(* Schneider Machine Expert - Basic project Timer New, file version 1.7.0.0 *)
(* ProjectInformations: Name=New project *)

HARDWARE
  Cpu 0: TM221M16R/G
  EthernetConfiguration: NetworkName=M221, IpAllocationMode=FixedAddress, IpAddress=0.0.0.0, SubnetMask=0.0.0.0
  SerialLineConfiguration: Baud=Baud19200, Parity=ParityEven, DataBits=DataBits8, StopBits=StopBits1, PhysicalMedium=PhysicalMediumRs485, TransmissionMode=TransmissionModeModbusRtu, SlaveId=1, Addressing=SlaveAddressing
  MastTask: UsePeriodScanMode=false, PeriodScan=100
  FastTask: Period=255
  CpuBehavior: StartingMode=StartAsPreviousState, AutoSaveRamOnEeprom=true, WatchdogPeriod=250

SYMBOLS  (address, symbol, comment, settings)
  %TM0        "T1"  [Preset=1, Base=OneSecond]
  %TM1        "T2"  [Preset=1, Base=OneSecond]
  %TM2        "T3"  [Preset=1, Base=OneSecond]
  %TM3        "T4"  [Preset=1, Base=OneSecond]
  %TM4        "TM5"  [Preset=1, Base=OneSecond]
  %TM5        "TM6"  [Preset=1, Base=OneSecond]
  %TM6        "TM7"  [Preset=1, Base=OneSecond]
  %TM7        "T8"  [Preset=1, Base=OneSecond]
  %I0.0       "Auto"
  %Q0.0       "L1"
  %Q0.1       "L2"
  %Q0.2       "L3"
  %Q0.3       "L4"

POU New POU
  (* SectionNumber=1 *)

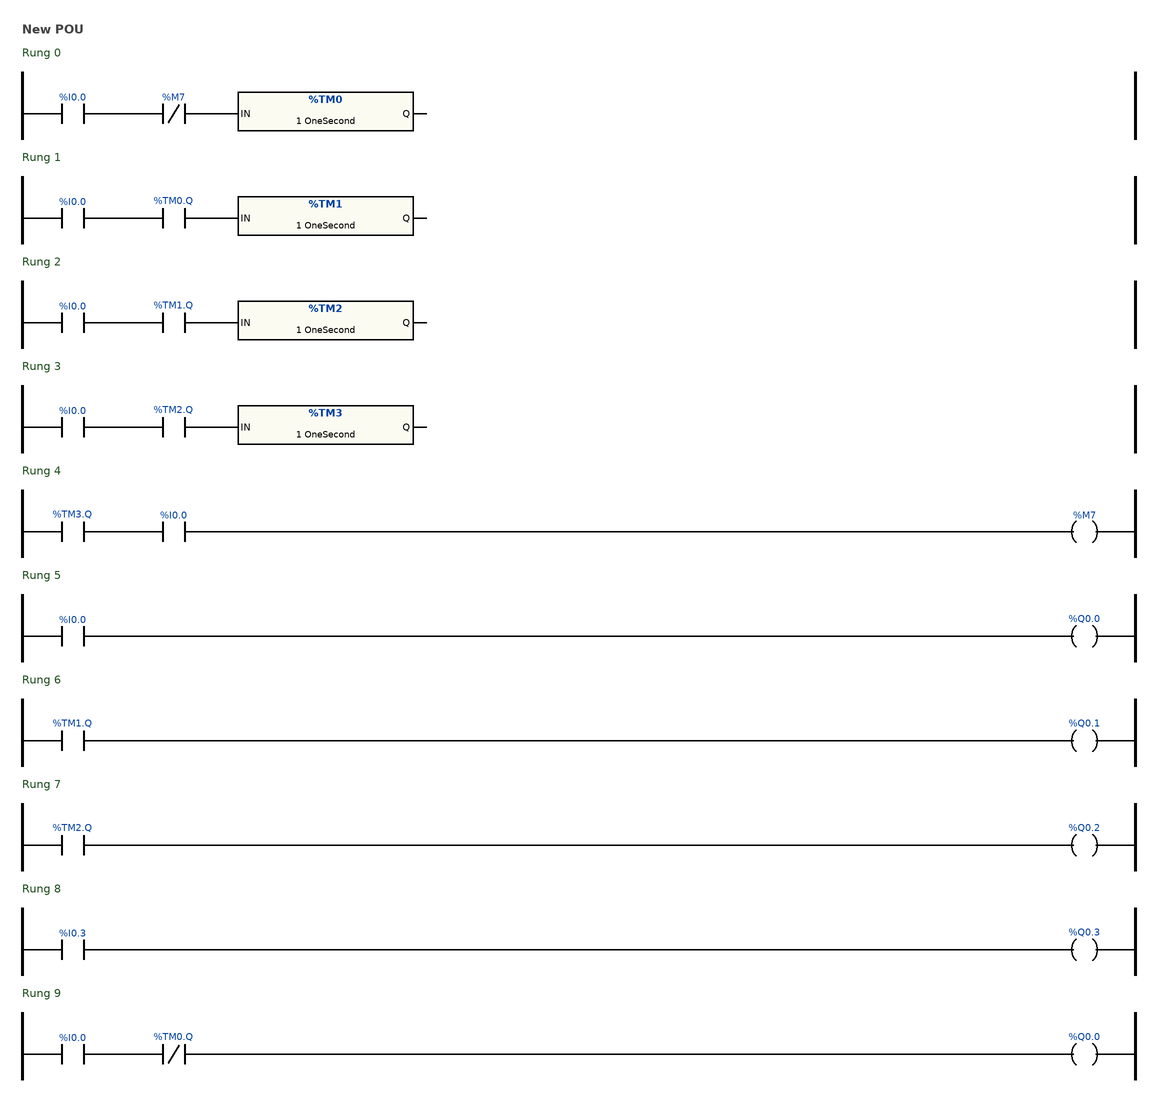

// Rung 0
  BLK %TM0
  LD %I0.0
  ANDN %M7
  IN
  END_BLK
  // as ST:
  //   %TM0(IN := %I0.0 AND NOT %M7);

// Rung 1
  BLK %TM1
  LD %I0.0
  AND %TM0.Q
  IN
  END_BLK
  // as ST:
  //   %TM1(IN := %I0.0 AND %TM0.Q);

// Rung 2
  BLK %TM2
  LD %I0.0
  AND %TM1.Q
  IN
  END_BLK
  // as ST:
  //   %TM2(IN := %I0.0 AND %TM1.Q);

// Rung 3
  BLK %TM3
  LD %I0.0
  AND %TM2.Q
  IN
  END_BLK
  // as ST:
  //   %TM3(IN := %I0.0 AND %TM2.Q);

// Rung 4
  LD %TM3.Q
  AND %I0.0
  ST %M7
  // as ST:
  //   %M7 := %TM3.Q AND %I0.0;

// Rung 5
  LD %I0.0
  ST %Q0.0
  // as ST:
  //   %Q0.0 := %I0.0;

// Rung 6
  LD %TM1.Q
  ST %Q0.1
  // as ST:
  //   %Q0.1 := %TM1.Q;

// Rung 7
  LD %TM2.Q
  ST %Q0.2
  // as ST:
  //   %Q0.2 := %TM2.Q;

// Rung 8
  LD %I0.3
  ST %Q0.3
  // as ST:
  //   %Q0.3 := %I0.3;

// Rung 9
  LD %I0.0
  ANDN %TM0.Q
  ST %Q0.0
  // as ST:
  //   %Q0.0 := %I0.0 AND NOT %TM0.Q;

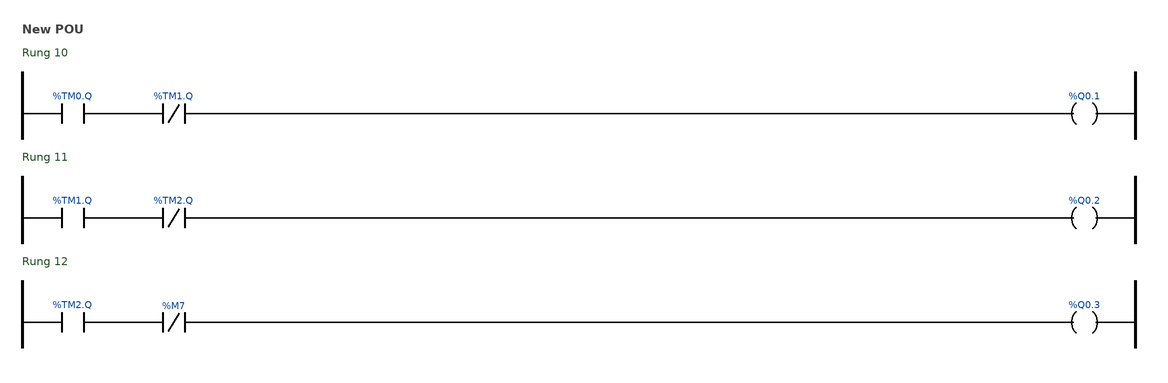

// Rung 10
  LD %TM0.Q
  ANDN %TM1.Q
  ST %Q0.1
  // as ST:
  //   %Q0.1 := %TM0.Q AND NOT %TM1.Q;

// Rung 11
  LD %TM1.Q
  ANDN %TM2.Q
  ST %Q0.2
  // as ST:
  //   %Q0.2 := %TM1.Q AND NOT %TM2.Q;

// Rung 12
  LD %TM2.Q
  ANDN %M7
  ST %Q0.3
  // as ST:
  //   %Q0.3 := %TM2.Q AND NOT %M7;
